Omron CX-Programmer project NewProject (CX-Programmer 9.50)

# PLC NewPLC1: CJ2M CPU34
I/O table (CPU CJ2M-CPU34): rack 0 slot 11 CJ2M-EIP21

## Global symbols (name address type ; comment)
Alignment D300 INT[10]  ; the alignment of each ballet with respect to the first ballet in the x axis
Assign_Pulse 11.00 BOOL
B_I_L D3 INT  ; number in boxes in layer selected by user
Box_angle D400 INT[40]  ; angle alignment of each box in the pallet
Dest_X D31 INT  ; final destination of the head for x axis
Dest_Y D32 INT  ; final destination of head in the y axis
Dest_Z D33 INT  ; final destination of the head in z axis
Destination D2 INT  ; no of pallet assigned to recive the boxes
Head_Angle D34 INT  ; destination angle of the current box
Last_box_code D0 INT  ; box ready to be gripped
Layer_No D900 INT[10]  ; no.of the layers in use in each pallet
Mach_Full D89 INT  ; alarm that the machine is full
N D1 INT  ; no. of pallets exist
No_Layer D36 INT  ; number of layer selected by user
Not_Assigned D30 INT  ; number to check that all pallets are not assigned with the current box type
P_code D600 INT[10]  ; pallet sorting code (1 small or big, 2 small or big, 3 small or big)
P_status D700 INT[10]  ; pallet status (active, diabled, full, no pallet)
Pos_X D100 INT[40]  ; position for each box in the x axis
Pos_Y D200 INT[40]  ; position for each box in the y axis
Pos_Z D90 INT[8]  ; position of each layer hieght in z axis
Ready_Pulse 11.02 BOOL
busy D4 INT
count D500 INT[10]  ; the amount of boxes in the ballet selected

## Program NewProgram1 (cyclic task 0)

### Section Section1

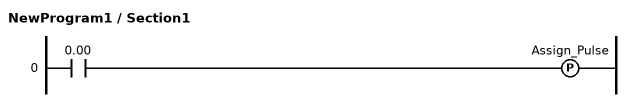
; rung 0
LD 0.00
DIFU(013) Assign_Pulse

### Section END
; rung 0
END(001)

## Program Assign_routine (cyclic task 1)
IF(Assign_Pulse= TRUE)THEN
	Not_Assigned:=0;
	FOR N:= 1 TO 9 DO
		IF (P_code[N]=Last_box_code AND P_status[N]=99)THEN
			Destination:=N;
			Ready_Pulse:= TRUE;
			EXIT;
		ELSE
			Not_Assigned:= Not_Assigned+1;
		END_IF;
	END_FOR;
	N:=1;
	busy:= 0;
	IF(Not_Assigned=9)THEN
		FOR N:= 1 TO 9 DO
			IF (P_status[N]=98)THEN
				Destination:=N;
				P_code[Destination]:=Last_box_code;
				Layer_No[Destination]:= 1;
				count[Destination]:= 0;
				P_status[Destination]:=99;
				Not_Assigned:=0;
				Ready_Pulse:=TRUE;
				EXIT;
			ELSE
				busy:=busy+1;
				IF(busy=9)THEN
				 Mach_Full:=1;
				END_IF;
			END_IF;
		END_FOR;
	END_IF;
END_IF;

## Program destination_routine (cyclic task 2)
IF (Ready_Pulse=TRUE)THEN
	IF (Layer_No[Destination]=1 OR Layer_No[Destination]= 3 OR Layer_No[Destination]= 5 OR Layer_No[Destination]= 7)THEN
		Dest_Z:= Pos_Z[Layer_No[Destination]];
		Dest_X:= Pos_X[count[Destination]+1] + Alignment[Destination];
		Dest_Y:= Pos_Y[count[Destination]+1];
		Head_Angle:= Box_angle[count[Destination]+1];
		count[Destination]:= count[Destination]+1;
	ELSIF (Layer_No[Destination]=2 OR Layer_No[Destination]= 4 OR Layer_No[Destination]= 6)THEN
		Dest_Z:= Pos_Z[Layer_No[Destination]];
		Dest_X:= Pos_X[ count[Destination] + B_I_L+1 ] + Alignment[Destination];
		Dest_Y:= Pos_Y[ count[Destination] + B_I_L +1];
		Head_Angle:= Box_angle[ count[Destination] + B_I_L+1 ];
		count[Destination]:= count[Destination]+1;
	END_IF;
	 IF (count[Destination]=B_I_L AND Layer_No[Destination]<No_Layer )THEN
		 Layer_No[Destination]:= Layer_No[Destination]+1;
		 count[Destination]:= 0;
	 ELSIF(Layer_No[Destination]=No_Layer AND count[Destination]=B_I_L)THEN
		  P_code[Destination]:= 0;
		  P_status[Destination]:=97;
		  count[Destination]:= 0;
	 END_IF;
END_IF;
Ready_Pulse:=FALSE;